TYPE MC_CAM_REF :
STRUCT
END_STRUCT
END_TYPE

(* stored: Version 1.1.0.1, ProductVersion 3.1.4024.12
   DUT MC_CAM_REF: Id {99e56ae5-6072-4aa3-83bd-13727c2c1e01} *)
